Staubli VAL3: place.pgx

program place(num x_nX, num x_nY)
begin



  pPlace.trsf.x = x_nX*100
  pPlace.trsf.y = x_nY*100

  movej(appro(pPlace,trApro),tGreifer, mUsedSpeed)
  movel(pPlace, tGreifer, mUsedSpeed)
  open(tGreifer)
  movel(appro(pPlace, trApro), tGreifer, mUsedSpeed)
  logMsg("Objekt abgelegt")





end
